INTERFACE I_DomainProvider EXTENDS I_Component

PROPERTY Self : I_Domain
GET
END_GET
END_PROPERTY

END_INTERFACE

(* stored: Version 1.1.0.1
   Itf I_DomainProvider: Id {b881675a-bfcc-4bda-b695-fb9178a5dfb4}
   Property Self: Id {abe5ce9a-2b0c-48f6-b54d-ef5937aaea34}
   Get Get: Id {b7b695ba-9ec8-43ce-af64-3471a08cee94} *)
